// TIA Portal V16 export
// export: Created 2025-08-30T12:59:11.3176565Z, ExportSetting WithDefaults, DisplayName Totally Integrated Automation Portal, DisplayVersion V16, DisplayName TIA Portal Version Control Interface, DisplayVersion V16, DisplayName TIA Portal Openness, DisplayVersion V16, DisplayName STEP 7 Professional, DisplayVersion V16, DisplayName STEP 7 Safety, DisplayVersion V16, DisplayName WinCC Advanced, DisplayVersion V16
FUNCTION "Axis_Confirmation" : Void   // FC7, FBD
TITLE = Axis Confirmation Block
VERSION : 0.1
// stored: AutoNumber true, IsIECCheckEnabled false, UDAEnableTagReadback false
   VAR_INPUT
      "Set Position" : Real;
   END_VAR
   VAR_OUTPUT
      "Axis On Position" : Bool;
      Min_Position_1 : Real;
      Max_Position_1 : Real;
   END_VAR
BEGIN

REGION Network 2: Calculate Position Tolerance 1
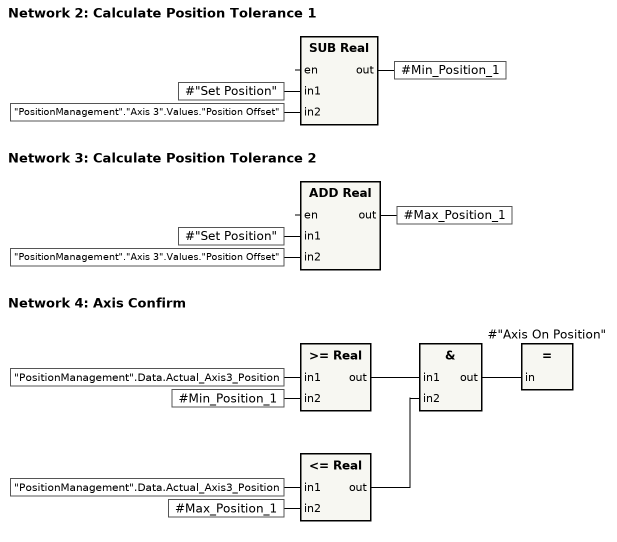
   #Min_Position_1 := #"Set Position" - "PositionManagement"."Axis 3".Values."Position Offset";
END_REGION

REGION Network 3: Calculate Position Tolerance 2
   #Max_Position_1 := #"Set Position" + "PositionManagement"."Axis 3".Values."Position Offset";
END_REGION

REGION Network 4: Axis Confirm
   #"Axis On Position" := ("PositionManagement".Data.Actual_Axis3_Position >= #Min_Position_1) AND ("PositionManagement".Data.Actual_Axis3_Position <= #Max_Position_1);
END_REGION
END_FUNCTION
